//{attribute 'qualified_only'}
VAR_GLOBAL
	fbPist:  ARRAY[1..30] OF FB_PIST;
END_VAR

(* stored: Version 1.1.0.1, ProductVersion 3.1.4024.12
   GVL GVL_PIST: Id {355e3a0f-01dd-4caf-8ab7-c00715794fa7} *)
